Fanuc KAREL source: ka00001.KL

-- PROVISIONAL review KL for V770-1; original PC SHA256 4110d2199f58eacea04ad418fd49075b7111edec18464f1f1c98e222829d8b80
-- Incomplete behavior may be omitted. Consult companion uncertainty JSON. Do not deploy.
PROGRAM KA00001
%NOLOCKGROUP
VAR
  SRC : INTEGER
  DST : INTEGER
BEGIN
  -- UNRESOLVED_PC offsets 5-16; opcodes 2E,23
  -- UNRESOLVED_PC offsets 21-33; opcodes 21,23
  -- UNRESOLVED_PC offsets 38-42; opcodes 7F
END KA00001
